FUNCTION F_LogA9 
VAR_INPUT
	eLogLevel		: E_LogLevel;
	sMessage		: T_MaxString;
	aArg1			: ANY;
	aArg2			: ANY;
	aArg3			: ANY;
	aArg4			: ANY;
	aArg5			: ANY;
	aArg6			: ANY;
	aArg7			: ANY;
	aArg8			: ANY;
	aArg9			: ANY;
END_VAR

F_LogLA9(eLogLevel, Const.sGlobalLogger, sMessage, aArg1, aArg2, aArg3, aArg4, aArg5, aArg6, aArg7, aArg8, aArg9);

END_FUNCTION

(* stored: Version 1.1.0.1, ProductVersion 3.1.4024.6
   POU F_LogA9: Id {427cd8e4-358a-4401-af05-ccc0e202c469}, SpecialFunc None *)
